FUNCTION FUN_ConvTwoByteToInt16 : INT
VAR_INPUT
	nValue1		:BYTE;				// Input Byte no 1
	nValue2		:BYTE;				// Input Byte no 2
END_VAR
VAR
	uData		:U_Convert_INT16;		// Data variable used for conversion
END_VAR


// Save input bytes in data union
uData.arrByte[1] := nValue1;
uData.arrByte[2] := nValue2;

// Return value
FUN_ConvTwoByteToInt16 := uData.nValue;

END_FUNCTION

(* stored: Version 1.1.0.1, ProductVersion 3.1.4024.12
   POU FUN_ConvTwoByteToInt16: Id {5cf9b8df-b64c-469c-b68a-154c5cae1636}, SpecialFunc None *)
